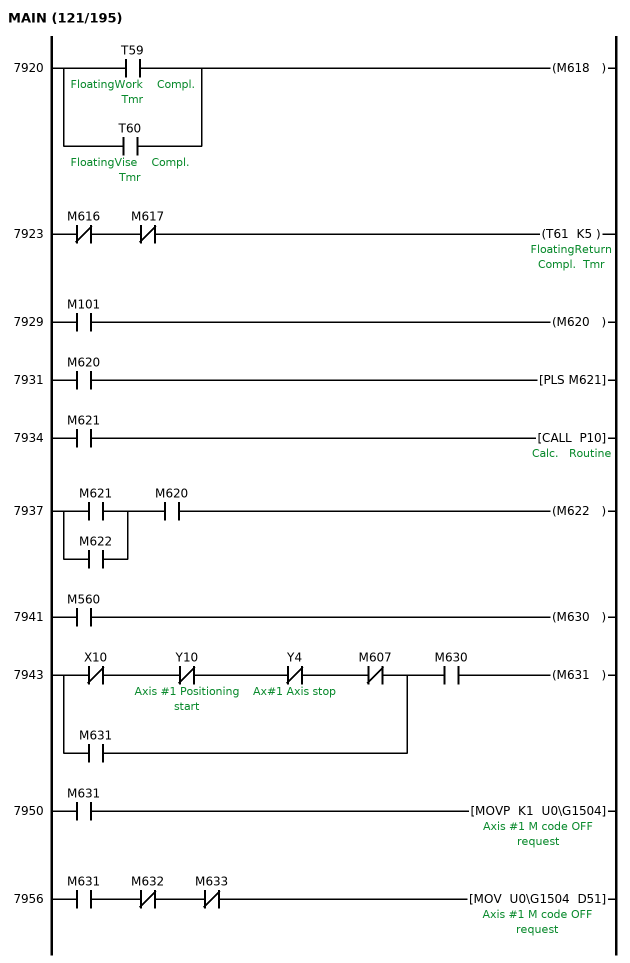
[picture p120: ladder of MAIN, rungs at steps 7920 to 7956]
7920  LD      T59  ; FloatingWork    Compl.  Tmr
      OR      T60  ; FloatingVise    Compl.  Tmr
      OUT     M618
7923  LDI     M616
      ANI     M617
      OUT     T61 K5  ; FloatingReturn  Compl.  Tmr
7929  LD      M101
      OUT     M620
7931  LD      M620
      PLS     M621
7934  LD      M621
      CALL    P10  ; Calc.   Routine
7937  LD      M621
      OR      M622
      AND     M620
      OUT     M622
7941  LD      M560
      OUT     M630
7943  LDI     X10
      ANI     Y10  ; Axis #1 Positioning start
      ANI     Y4  ; Ax#1 Axis stop
      ANI     M607
      OR      M631
      AND     M630
      OUT     M631
7950  LD      M631
      MOVP    K1 U0\G1504  ; Axis #1 M code OFF request
7956  LD      M631
      ANI     M632
      ANI     M633
      MOV     U0\G1504 D51
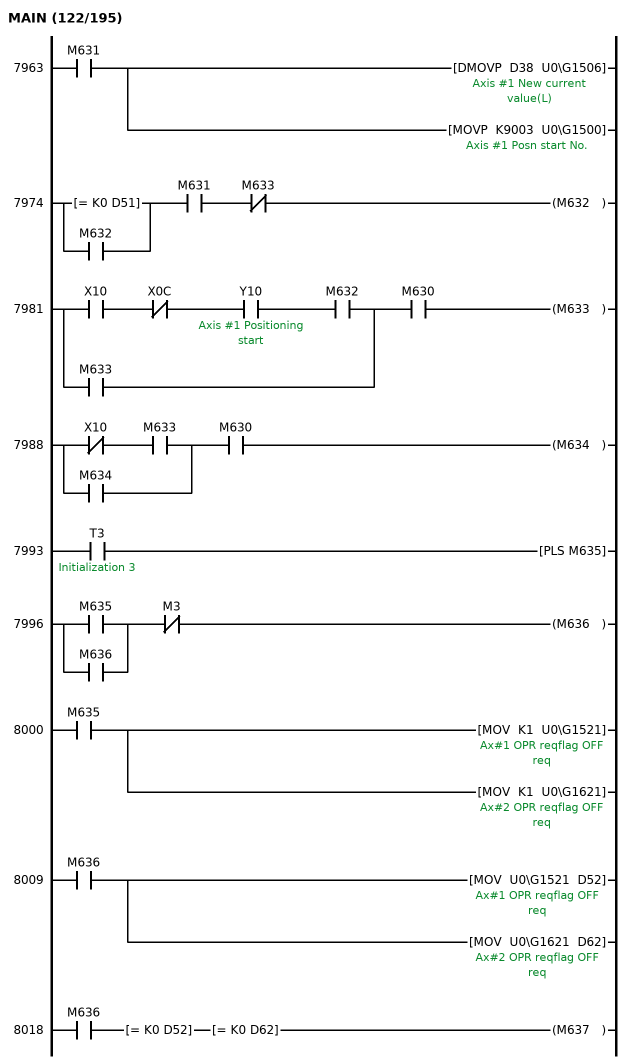
7963  LD      M631
      DMOVP   D38 U0\G1506  ; Axis #1 New current value(L)
      MOVP    K9003 U0\G1500
7974  LD=     K0 D51
      OR      M632
      AND     M631
      ANI     M633
      OUT     M632
7981  LD      X10
      ANI     X0C
      AND     Y10  ; Axis #1 Positioning start
      AND     M632
      OR      M633
      AND     M630
      OUT     M633
7988  LDI     X10
      AND     M633
      OR      M634
      AND     M630
      OUT     M634
7993  LD      T3  ; Initialization 3
      PLS     M635
7996  LD      M635
      OR      M636
      ANI     M3
      OUT     M636
8000  LD      M635
      MOV     K1 U0\G1521  ; Ax#1 OPR reqflag OFF req
      MOV     K1 U0\G1621  ; Ax#2 OPR reqflag OFF req
8009  LD      M636
      MOV     U0\G1521 D52
      MOV     U0\G1621 D62
8018  LD      M636
      AND=    K0 D52
      AND=    K0 D62
      OUT     M637
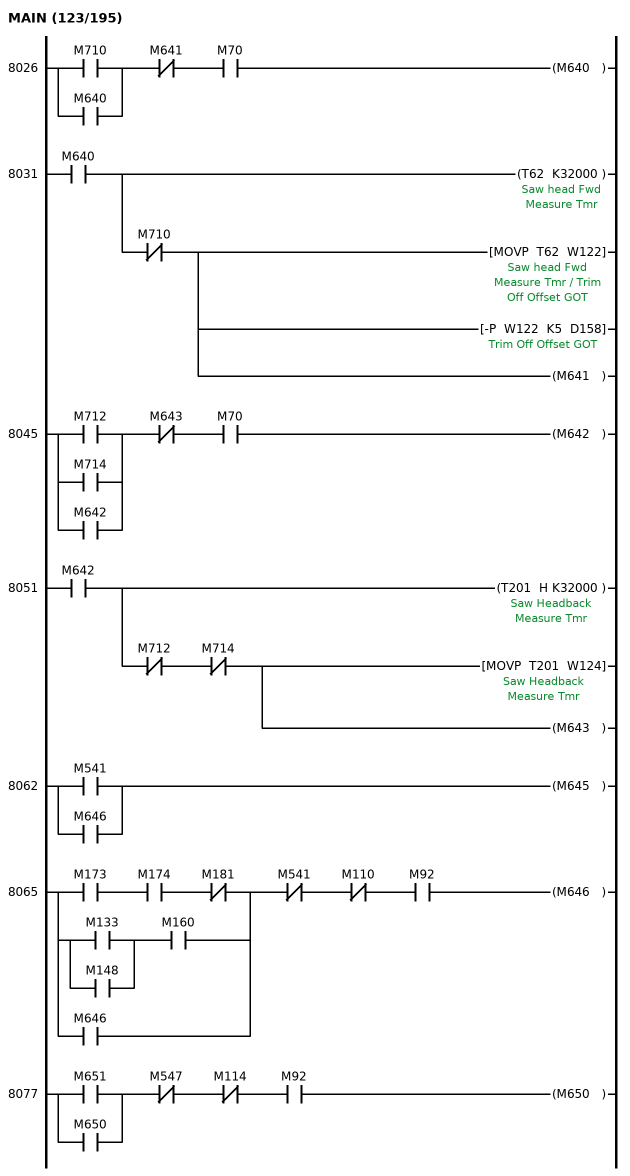
8026  LD      M710
      OR      M640
      ANI     M641
      AND     M70
      OUT     M640
8031  LD      M640
      OUT     T62 K32000  ; Saw head Fwd    Measure Tmr
      ANI     M710
      MOVP    T62 W122  ; Trim Off Offset GOT
      -P      W122 K5 D158
      OUT     M641
8045  LD      M712
      OR      M714
      OR      M642
      ANI     M643
      AND     M70
      OUT     M642
8051  LD      M642
      OUTH    T201 K32000  ; Saw Headback    Measure Tmr
      ANI     M712
      ANI     M714
      MOVP    T201 W124
      OUT     M643
8062  LD      M541
      OR      M646
      OUT     M645
8065  LD      M173
      AND     M174
      ANI     M181
      LD      M133
      OR      M148
      AND     M160
      ORB
      OR      M646
      ANI     M541
      ANI     M110
      AND     M92
      OUT     M646
8077  LD      M651
      OR      M650
      ANI     M547
      ANI     M114
      AND     M92
      OUT     M650
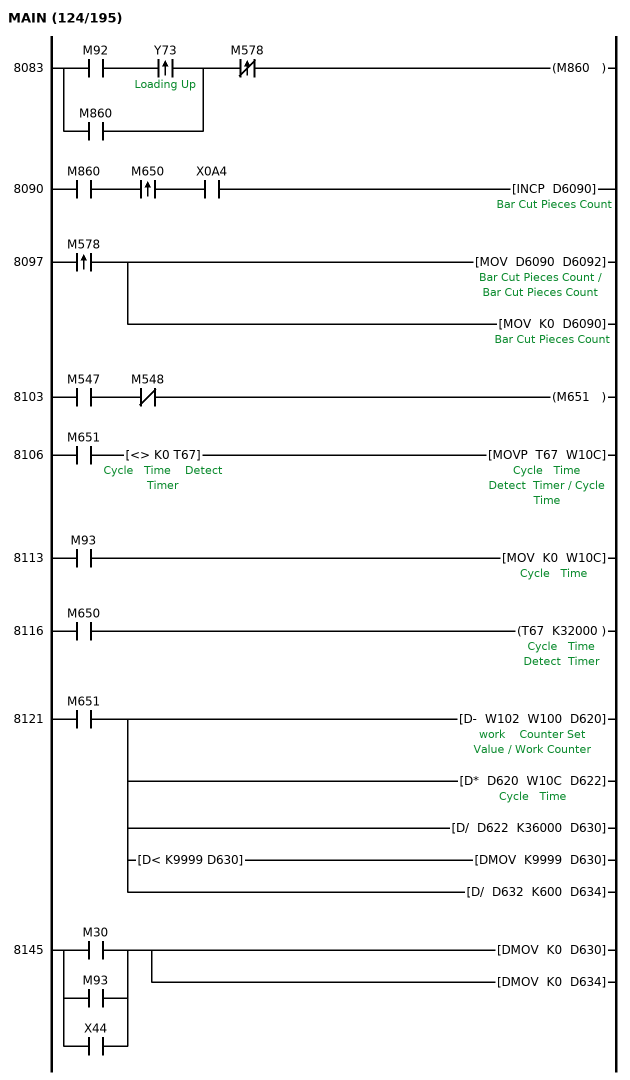
8083  LD      M92
      ANDP    Y73  ; Loading Up
      OR      M860
      ANDPI   M578
      OUT     M860
8090  LD      M860
      ANDP    M650
      AND     X0A4
      INCP    D6090  ; Bar Cut Pieces Count
8097  LDP     M578
      MOV     D6090 D6092  ; Bar Cut Pieces Count
      MOV     K0 D6090
8103  LD      M547
      ANI     M548
      OUT     M651
8106  LD      M651
      AND<>   K0 T67  ; Cycle   Time    Detect  Timer
      MOVP    T67 W10C  ; Cycle   Time
8113  LD      M93
      MOV     K0 W10C
8116  LD      M650
      OUT     T67 K32000  ; Cycle   Time    Detect  Timer
8121  LD      M651
      D-      W102 W100 D620
      D*      D620 W10C D622
      D/      D622 K36000 D630
      MPS
      ANDD<   K9999 D630
      DMOV    K9999 D630
      MPP
      D/      D632 K600 D634
8145  LD      M30
      OR      M93
      OR      X44
      DMOV    K0 D630
      DMOV    K0 D634
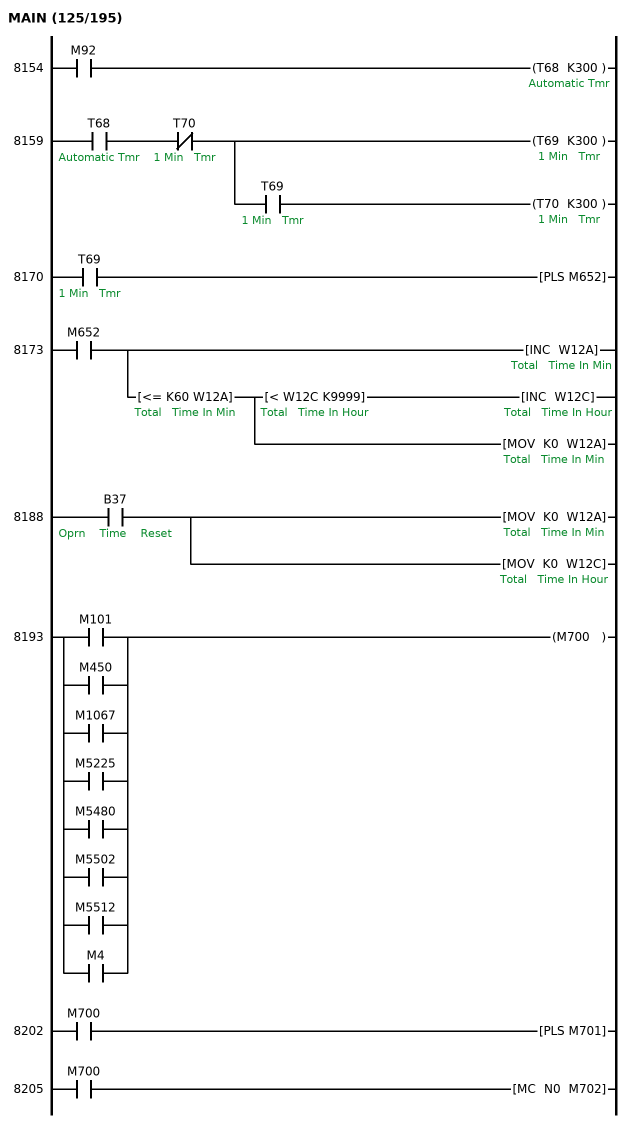
8154  LD      M92
      OUT     T68 K300  ; Automatic Tmr
8159  LD      T68  ; Automatic Tmr
      ANI     T70  ; 1 Min   Tmr
      OUT     T69 K300  ; 1 Min   Tmr
      AND     T69  ; 1 Min   Tmr
      OUT     T70 K300  ; 1 Min   Tmr
8170  LD      T69  ; 1 Min   Tmr
      PLS     M652
8173  LD      M652
      INC     W12A  ; Total   Time In Min
      AND<=   K60 W12A  ; Total   Time In Min
      MPS
      AND<    W12C K9999  ; Total   Time In Hour
      INC     W12C
      MPP
      MOV     K0 W12A
8188  LD      B37  ; Oprn    Time    Reset
      MOV     K0 W12A
      MOV     K0 W12C
8193  LD      M101
      OR      M450
      OR      M1067
      OR      M5225
      OR      M5480
      OR      M5502
      OR      M5512
      OR      M4
      OUT     M700
8202  LD      M700
      PLS     M701
8205  LD      M700
      MC      N0 M702
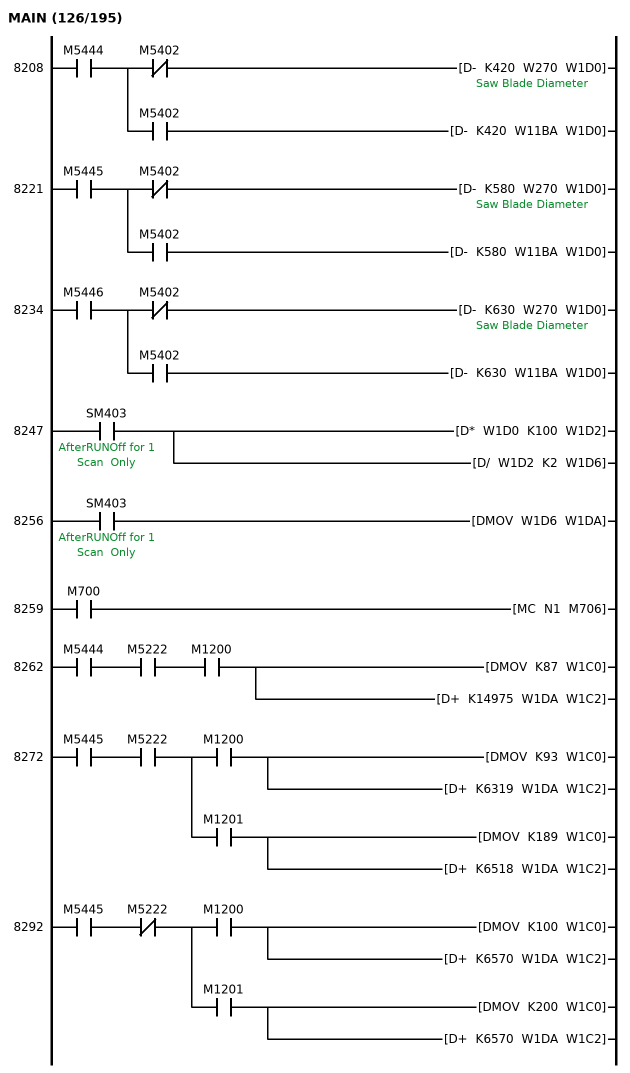
8208  LD      M5444
      MPS
      ANI     M5402
      D-      K420 W270 W1D0
      MPP
      AND     M5402
      D-      K420 W11BA W1D0
8221  LD      M5445
      MPS
      ANI     M5402
      D-      K580 W270 W1D0
      MPP
      AND     M5402
      D-      K580 W11BA W1D0
8234  LD      M5446
      MPS
      ANI     M5402
      D-      K630 W270 W1D0
      MPP
      AND     M5402
      D-      K630 W11BA W1D0
8247  LD      SM403  ; AfterRUNOff for 1 Scan  Only
      D*      W1D0 K100 W1D2
      D/      W1D2 K2 W1D6
8256  LD      SM403  ; AfterRUNOff for 1 Scan  Only
      DMOV    W1D6 W1DA
8259  LD      M700
      MC      N1 M706
8262  LD      M5444
      AND     M5222
      AND     M1200
      DMOV    K87 W1C0
      D+      K14975 W1DA W1C2
8272  LD      M5445
      AND     M5222
      MPS
      AND     M1200
      DMOV    K93 W1C0
      D+      K6319 W1DA W1C2
      MPP
      AND     M1201
      DMOV    K189 W1C0
      D+      K6518 W1DA W1C2
8292  LD      M5445
      ANI     M5222
      MPS
      AND     M1200
      DMOV    K100 W1C0
      D+      K6570 W1DA W1C2
      MPP
      AND     M1201
      DMOV    K200 W1C0
      D+      K6570 W1DA W1C2
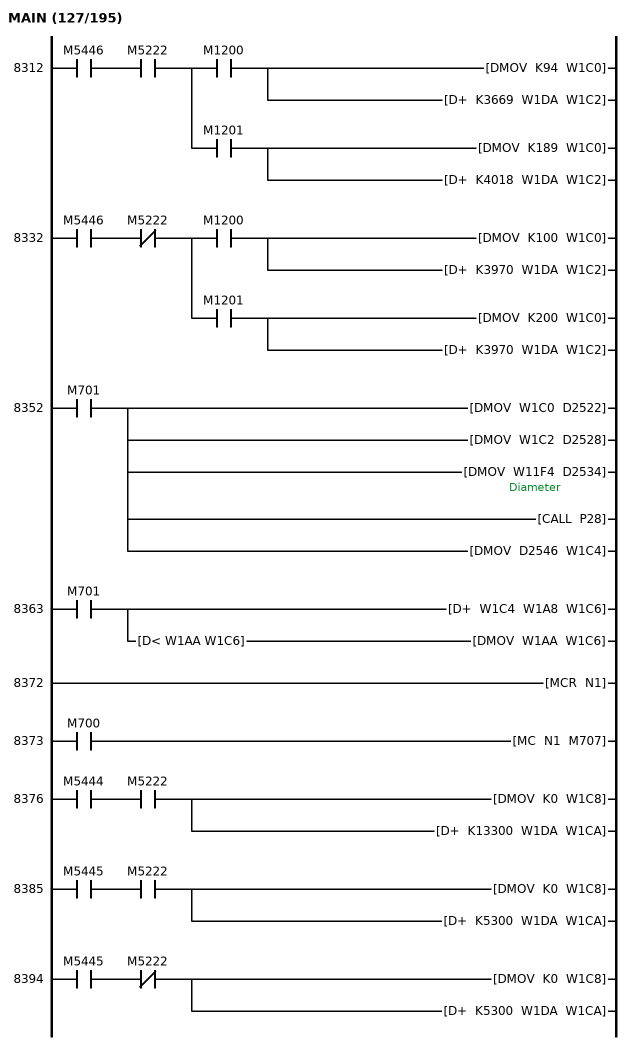
8312  LD      M5446
      AND     M5222
      MPS
      AND     M1200
      DMOV    K94 W1C0
      D+      K3669 W1DA W1C2
      MPP
      AND     M1201
      DMOV    K189 W1C0
      D+      K4018 W1DA W1C2
8332  LD      M5446
      ANI     M5222
      MPS
      AND     M1200
      DMOV    K100 W1C0
      D+      K3970 W1DA W1C2
      MPP
      AND     M1201
      DMOV    K200 W1C0
      D+      K3970 W1DA W1C2
8352  LD      M701
      DMOV    W1C0 D2522
      DMOV    W1C2 D2528
      DMOV    W11F4 D2534
      CALL    P28
      DMOV    D2546 W1C4
8363  LD      M701
      D+      W1C4 W1A8 W1C6
      ANDD<   W1AA W1C6
      DMOV    W1AA W1C6
8372  MCR     N1
8373  LD      M700
      MC      N1 M707
8376  LD      M5444
      AND     M5222
      DMOV    K0 W1C8
      D+      K13300 W1DA W1CA
8385  LD      M5445
      AND     M5222
      DMOV    K0 W1C8
      D+      K5300 W1DA W1CA
8394  LD      M5445
      ANI     M5222
      DMOV    K0 W1C8
      D+      K5300 W1DA W1CA
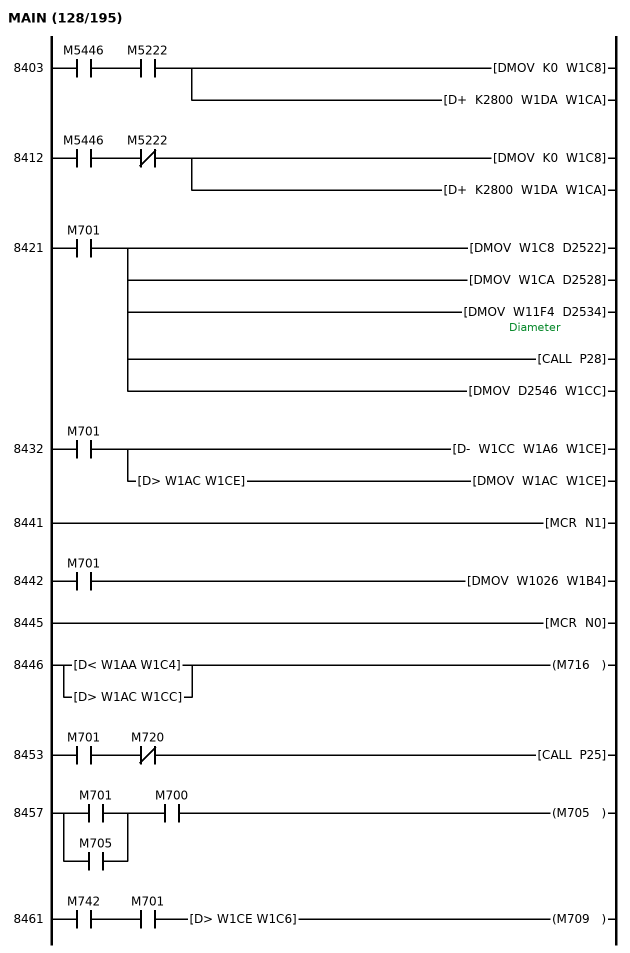
8403  LD      M5446
      AND     M5222
      DMOV    K0 W1C8
      D+      K2800 W1DA W1CA
8412  LD      M5446
      ANI     M5222
      DMOV    K0 W1C8
      D+      K2800 W1DA W1CA
8421  LD      M701
      DMOV    W1C8 D2522
      DMOV    W1CA D2528
      DMOV    W11F4 D2534
      CALL    P28
      DMOV    D2546 W1CC
8432  LD      M701
      D-      W1CC W1A6 W1CE
      ANDD>   W1AC W1CE
      DMOV    W1AC W1CE
8441  MCR     N1
8442  LD      M701
      DMOV    W1026 W1B4
8445  MCR     N0
8446  LDD<    W1AA W1C4
      ORD>    W1AC W1CC
      OUT     M716
8453  LD      M701
      ANI     M720
      CALL    P25
8457  LD      M701
      OR      M705
      AND     M700
      OUT     M705
8461  LD      M742
      AND     M701
      ANDD>   W1CE W1C6
      OUT     M709
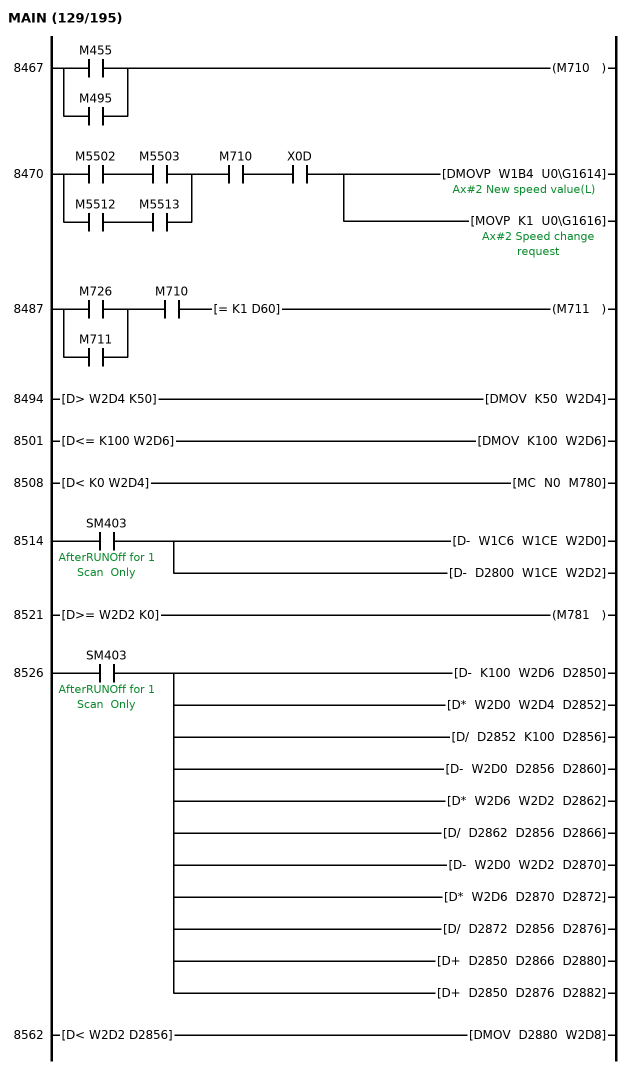
8467  LD      M455
      OR      M495
      OUT     M710
8470  LD      M5502
      AND     M5503
      LD      M5512
      AND     M5513
      ORB
      AND     M710
      AND     X0D
      DMOVP   W1B4 U0\G1614  ; Ax#2 New speed value(L)
      MOVP    K1 U0\G1616  ; Ax#2 Speed change request
8487  LD      M726
      OR      M711
      AND     M710
      AND=    K1 D60
      OUT     M711
8494  LDD>    W2D4 K50
      DMOV    K50 W2D4
8501  LDD<=   K100 W2D6
      DMOV    K100 W2D6
8508  LDD<    K0 W2D4
      MC      N0 M780
8514  LD      SM403  ; AfterRUNOff for 1 Scan  Only
      D-      W1C6 W1CE W2D0
      D-      D2800 W1CE W2D2
8521  LDD>=   W2D2 K0
      OUT     M781
8526  LD      SM403  ; AfterRUNOff for 1 Scan  Only
      D-      K100 W2D6 D2850
      D*      W2D0 W2D4 D2852
      D/      D2852 K100 D2856
      D-      W2D0 D2856 D2860
      D*      W2D6 W2D2 D2862
      D/      D2862 D2856 D2866
      D-      W2D0 W2D2 D2870
      D*      W2D6 D2870 D2872
      D/      D2872 D2856 D2876
      D+      D2850 D2866 D2880
      D+      D2850 D2876 D2882
8562  LDD<    W2D2 D2856
      DMOV    D2880 W2D8
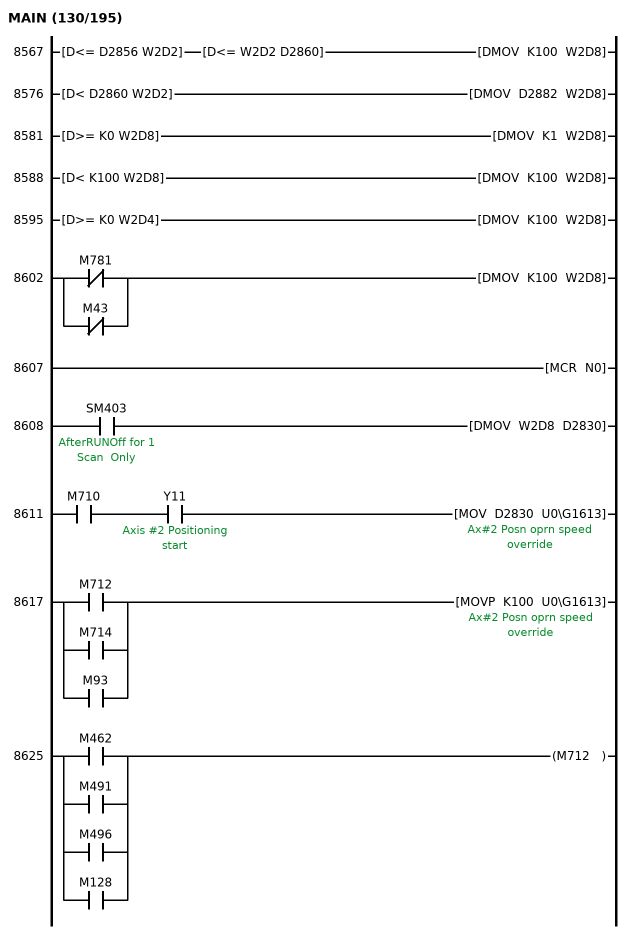
8567  LDD<=   D2856 W2D2
      ANDD<=  W2D2 D2860
      DMOV    K100 W2D8
8576  LDD<    D2860 W2D2
      DMOV    D2882 W2D8
8581  LDD>=   K0 W2D8
      DMOV    K1 W2D8
8588  LDD<    K100 W2D8
      DMOV    K100 W2D8
8595  LDD>=   K0 W2D4
      DMOV    K100 W2D8
8602  LDI     M781
      ORI     M43
      DMOV    K100 W2D8
8607  MCR     N0
8608  LD      SM403  ; AfterRUNOff for 1 Scan  Only
      DMOV    W2D8 D2830
8611  LD      M710
      AND     Y11  ; Axis #2 Positioning start
      MOV     D2830 U0\G1613  ; Ax#2 Posn oprn speed override
8617  LD      M712
      OR      M714
      OR      M93
      MOVP    K100 U0\G1613
8625  LD      M462
      OR      M491
      OR      M496
      OR      M128
      OUT     M712
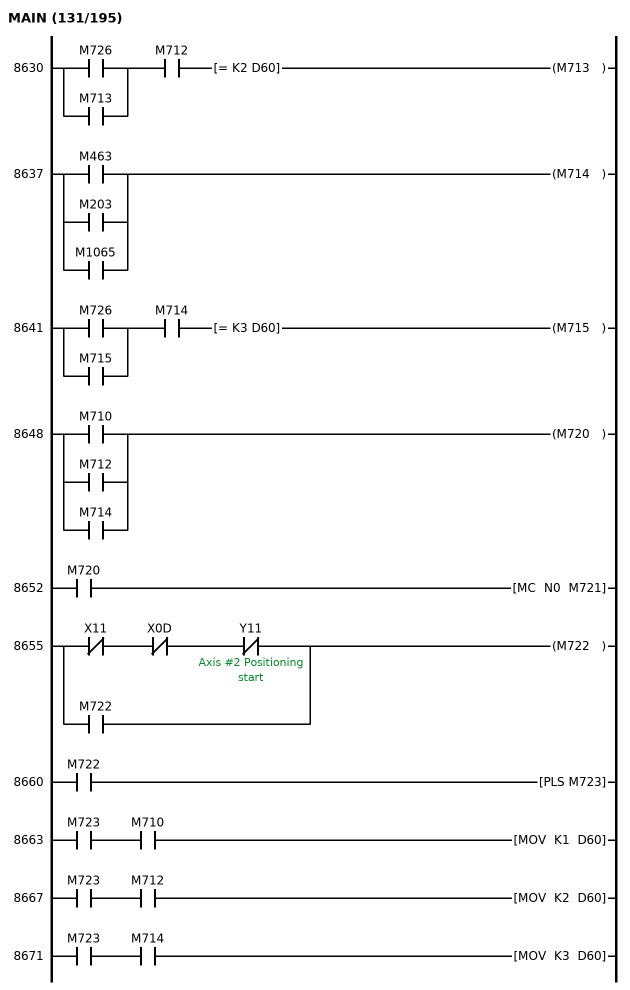
8630  LD      M726
      OR      M713
      AND     M712
      AND=    K2 D60
      OUT     M713
8637  LD      M463
      OR      M203
      OR      M1065
      OUT     M714
8641  LD      M726
      OR      M715
      AND     M714
      AND=    K3 D60
      OUT     M715
8648  LD      M710
      OR      M712
      OR      M714
      OUT     M720
8652  LD      M720
      MC      N0 M721
8655  LDI     X11
      ANI     X0D
      ANI     Y11  ; Axis #2 Positioning start
      OR      M722
      OUT     M722
8660  LD      M722
      PLS     M723
8663  LD      M723
      AND     M710
      MOV     K1 D60
8667  LD      M723
      AND     M712
      MOV     K2 D60
8671  LD      M723
      AND     M714
      MOV     K3 D60
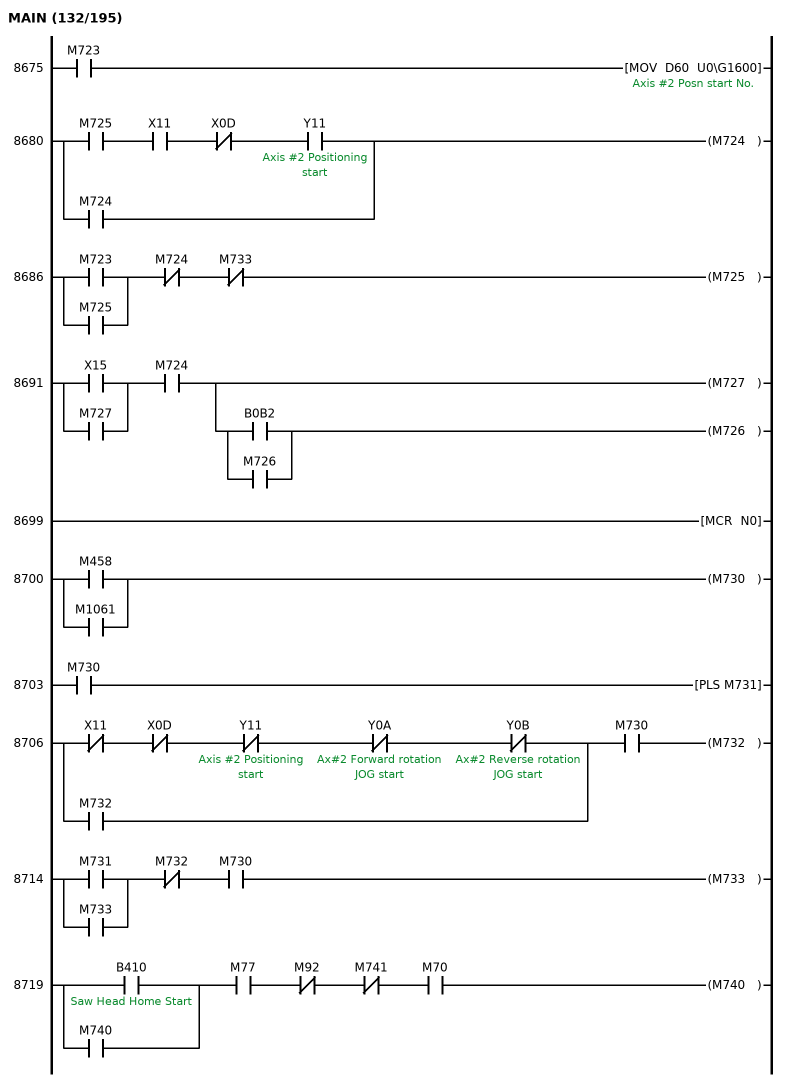
8675  LD      M723
      MOV     D60 U0\G1600  ; Axis #2 Posn start No.
8680  LD      M725
      AND     X11
      ANI     X0D
      AND     Y11  ; Axis #2 Positioning start
      OR      M724
      OUT     M724
8686  LD      M723
      OR      M725
      ANI     M724
      ANI     M733
      OUT     M725
8691  LD      X15
      OR      M727
      AND     M724
      OUT     M727
      LD      B0B2
      OR      M726
      ANB
      OUT     M726
8699  MCR     N0
8700  LD      M458
      OR      M1061
      OUT     M730
8703  LD      M730
      PLS     M731
8706  LDI     X11
      ANI     X0D
      ANI     Y11  ; Axis #2 Positioning start
      ANI     Y0A  ; Ax#2 Forward rotation JOG start
      ANI     Y0B  ; Ax#2 Reverse rotation JOG start
      OR      M732
      AND     M730
      OUT     M732
8714  LD      M731
      OR      M733
      ANI     M732
      AND     M730
      OUT     M733
8719  LD      B410  ; Saw Head Home Start
      OR      M740
      AND     M77
      ANI     M92
      ANI     M741
      AND     M70
      OUT     M740
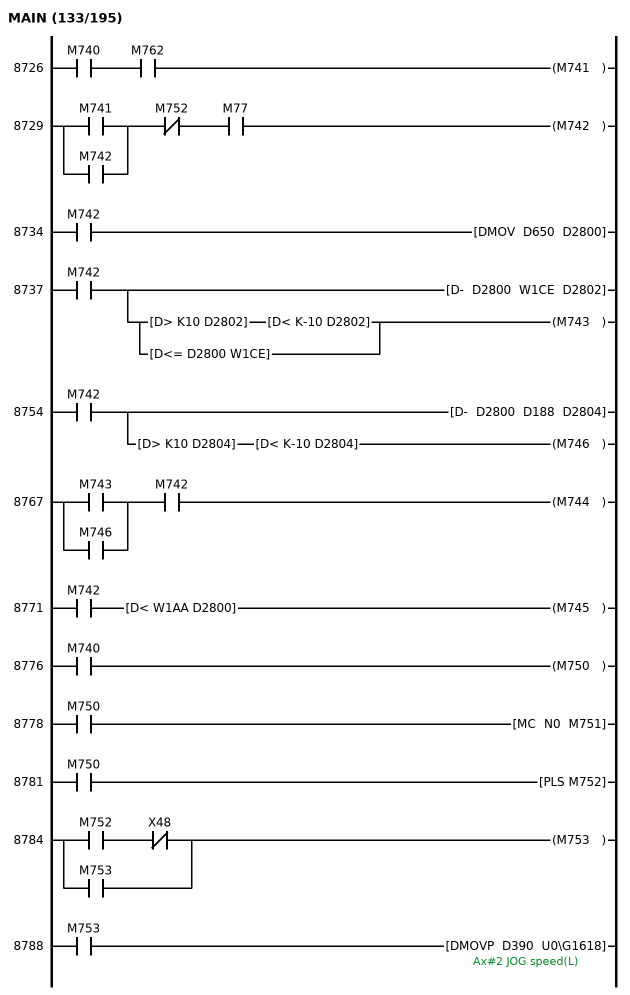
8726  LD      M740
      AND     M762
      OUT     M741
8729  LD      M741
      OR      M742
      ANI     M752
      AND     M77
      OUT     M742
8734  LD      M742
      DMOV    D650 D2800
8737  LD      M742
      D-      D2800 W1CE D2802
      LDD>    K10 D2802
      ANDD<   K-10 D2802
      ORD<=   D2800 W1CE
      ANB
      OUT     M743
8754  LD      M742
      D-      D2800 D188 D2804
      ANDD>   K10 D2804
      ANDD<   K-10 D2804
      OUT     M746
8767  LD      M743
      OR      M746
      AND     M742
      OUT     M744
8771  LD      M742
      ANDD<   W1AA D2800
      OUT     M745
8776  LD      M740
      OUT     M750
8778  LD      M750
      MC      N0 M751
8781  LD      M750
      PLS     M752
8784  LD      M752
      ANI     X48
      OR      M753
      OUT     M753
8788  LD      M753
      DMOVP   D390 U0\G1618
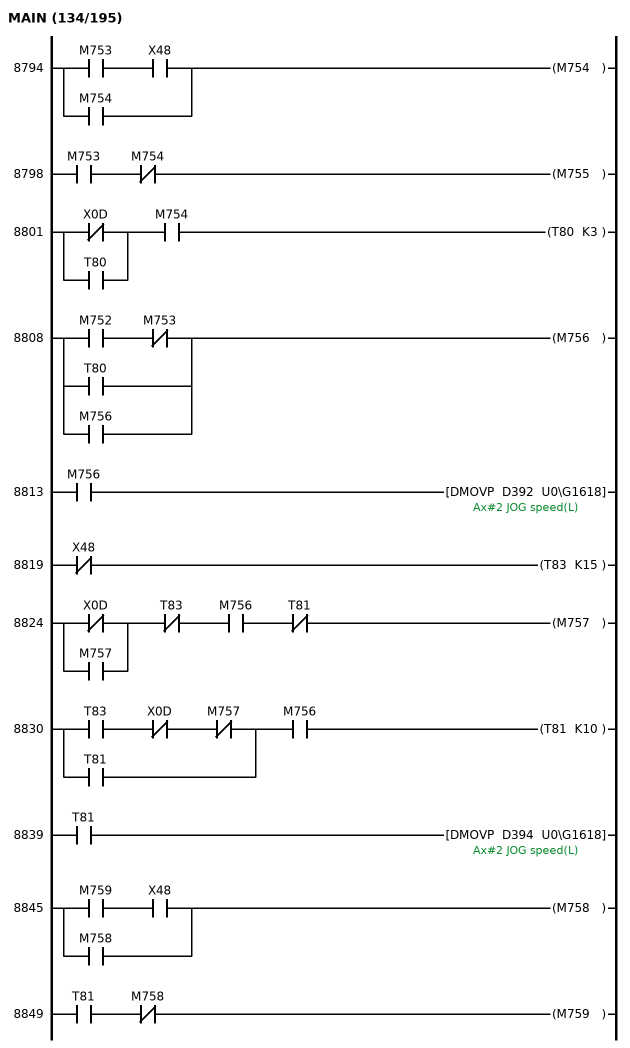
8794  LD      M753
      AND     X48
      OR      M754
      OUT     M754
8798  LD      M753
      ANI     M754
      OUT     M755
8801  LDI     X0D
      OR      T80
      AND     M754
      OUT     T80 K3
8808  LD      M752
      ANI     M753
      OR      T80
      OR      M756
      OUT     M756
8813  LD      M756
      DMOVP   D392 U0\G1618
8819  LDI     X48
      OUT     T83 K15
8824  LDI     X0D
      OR      M757
      ANI     T83
      AND     M756
      ANI     T81
      OUT     M757
8830  LD      T83
      ANI     X0D
      ANI     M757
      OR      T81
      AND     M756
      OUT     T81 K10
8839  LD      T81
      DMOVP   D394 U0\G1618
8845  LD      M759
      AND     X48
      OR      M758
      OUT     M758
8849  LD      T81
      ANI     M758
      OUT     M759
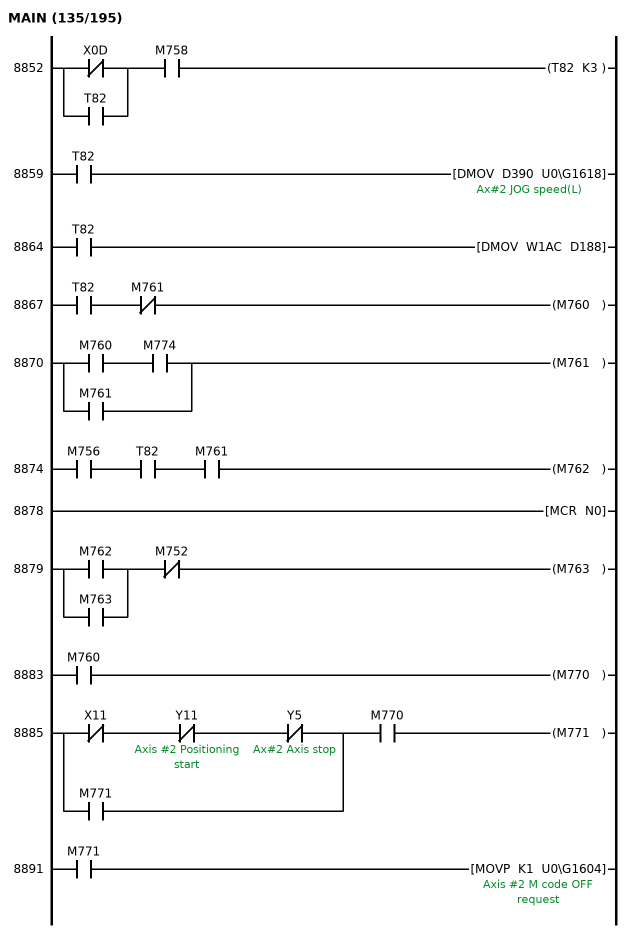
8852  LDI     X0D
      OR      T82
      AND     M758
      OUT     T82 K3
8859  LD      T82
      DMOV    D390 U0\G1618
8864  LD      T82
      DMOV    W1AC D188
8867  LD      T82
      ANI     M761
      OUT     M760
8870  LD      M760
      AND     M774
      OR      M761
      OUT     M761
8874  LD      M756
      AND     T82
      AND     M761
      OUT     M762
8878  MCR     N0
8879  LD      M762
      OR      M763
      ANI     M752
      OUT     M763
8883  LD      M760
      OUT     M770
8885  LDI     X11
      ANI     Y11  ; Axis #2 Positioning start
      ANI     Y5  ; Ax#2 Axis stop
      OR      M771
      AND     M770
      OUT     M771
8891  LD      M771
      MOVP    K1 U0\G1604  ; Axis #2 M code OFF request
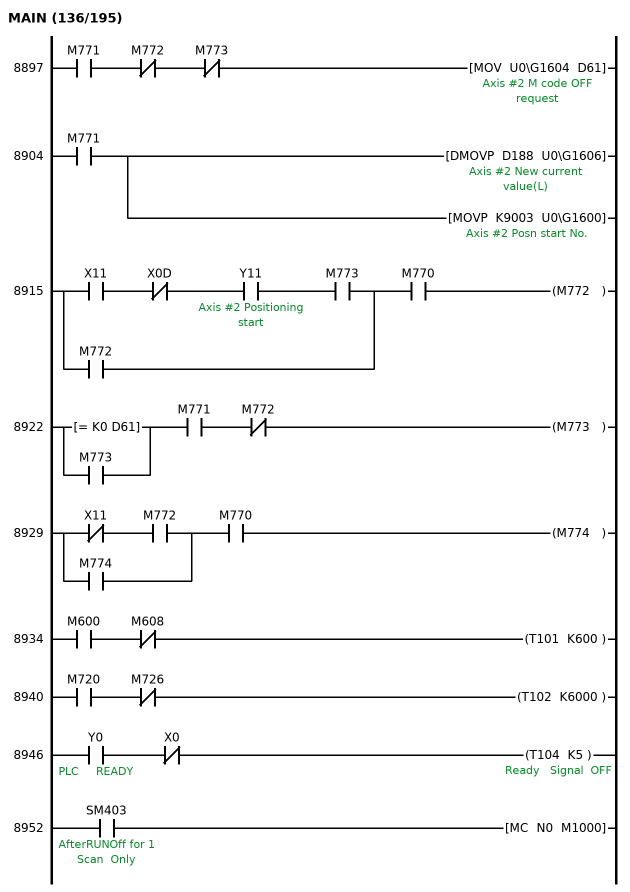
8897  LD      M771
      ANI     M772
      ANI     M773
      MOV     U0\G1604 D61
8904  LD      M771
      DMOVP   D188 U0\G1606  ; Axis #2 New current value(L)
      MOVP    K9003 U0\G1600
8915  LD      X11
      ANI     X0D
      AND     Y11  ; Axis #2 Positioning start
      AND     M773
      OR      M772
      AND     M770
      OUT     M772
8922  LD=     K0 D61
      OR      M773
      AND     M771
      ANI     M772
      OUT     M773
8929  LDI     X11
      AND     M772
      OR      M774
      AND     M770
      OUT     M774
8934  LD      M600
      ANI     M608
      OUT     T101 K600
8940  LD      M720
      ANI     M726
      OUT     T102 K6000
8946  LD      Y0  ; PLC     READY
      ANI     X0
      OUT     T104 K5  ; Ready   Signal  OFF
8952  LD      SM403  ; AfterRUNOff for 1 Scan  Only
      MC      N0 M1000
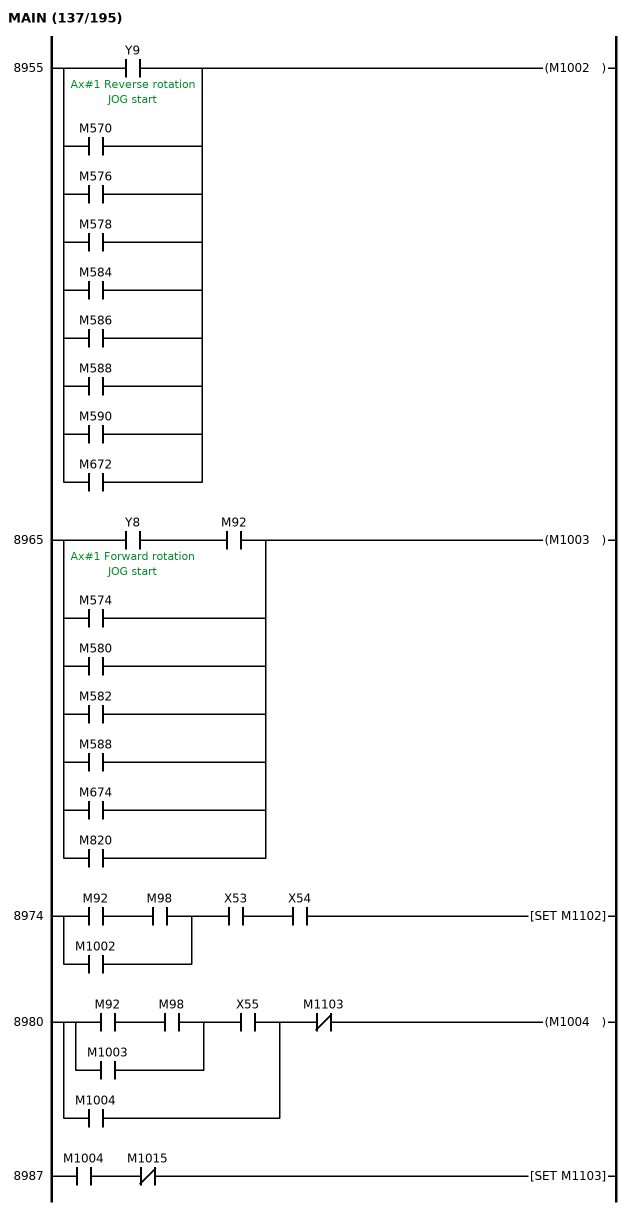
8955  LD      Y9  ; Ax#1 Reverse rotation JOG start
      OR      M570
      OR      M576
      OR      M578
      OR      M584
      OR      M586
      OR      M588
      OR      M590
      OR      M672
      OUT     M1002
8965  LD      Y8  ; Ax#1 Forward rotation JOG start
      AND     M92
      OR      M574
      OR      M580
      OR      M582
      OR      M588
      OR      M674
      OR      M820
      OUT     M1003
8974  LD      M92
      AND     M98
      OR      M1002
      AND     X53
      AND     X54
      SET     M1102
8980  LD      M92
      AND     M98
      OR      M1003
      AND     X55
      OR      M1004
      ANI     M1103
      OUT     M1004
8987  LD      M1004
      ANI     M1015
      SET     M1103
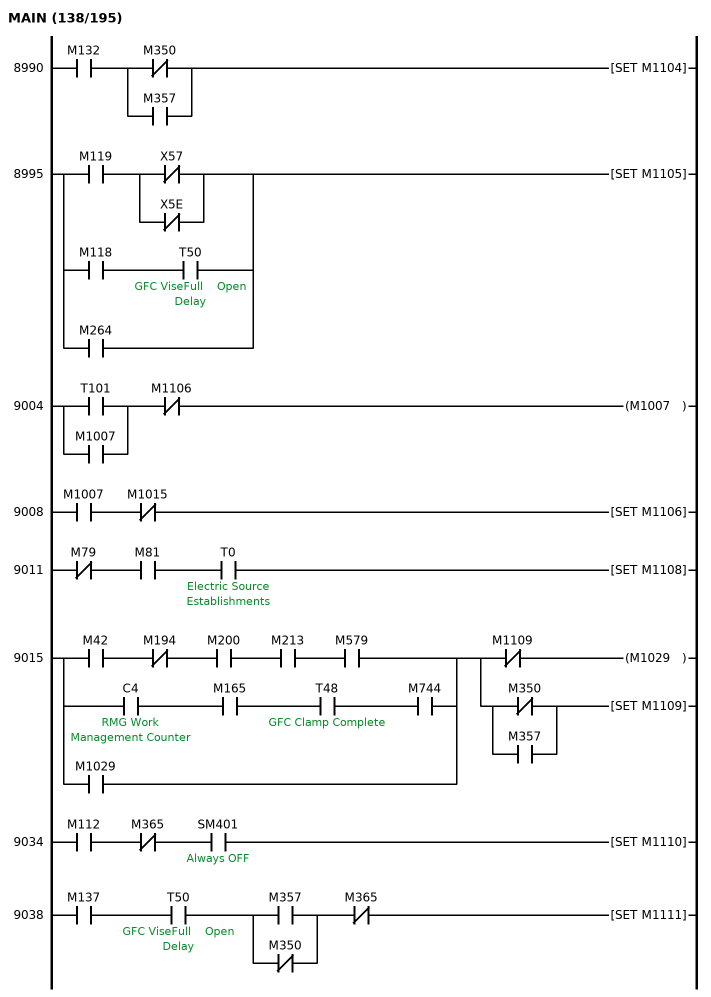
8990  LD      M132
      LDI     M350
      OR      M357
      ANB
      SET     M1104
8995  LD      M119
      LDI     X57
      ORI     X5E
      ANB
      LD      M118
      AND     T50  ; GFC ViseFull    Open    Delay
      ORB
      OR      M264
      SET     M1105
9004  LD      T101
      OR      M1007
      ANI     M1106
      OUT     M1007
9008  LD      M1007
      ANI     M1015
      SET     M1106
9011  LDI     M79
      AND     M81
      AND     T0  ; Electric Source Establishments
      SET     M1108
9015  LD      M42
      ANI     M194
      AND     M200
      AND     M213
      AND     M579
      LD      C4  ; RMG WorkManagement Counter
      AND     M165
      AND     T48  ; GFC Clamp Complete
      AND     M744
      ORB
      OR      M1029
      MPS
      ANI     M1109
      OUT     M1029
      MPP
      LDI     M350
      OR      M357
      ANB
      SET     M1109
9034  LD      M112
      ANI     M365
      AND     SM401  ; Always OFF
      SET     M1110
9038  LD      M137
      AND     T50  ; GFC ViseFull    Open    Delay
      LD      M357
      ORI     M350
      ANB
      ANI     M365
      SET     M1111
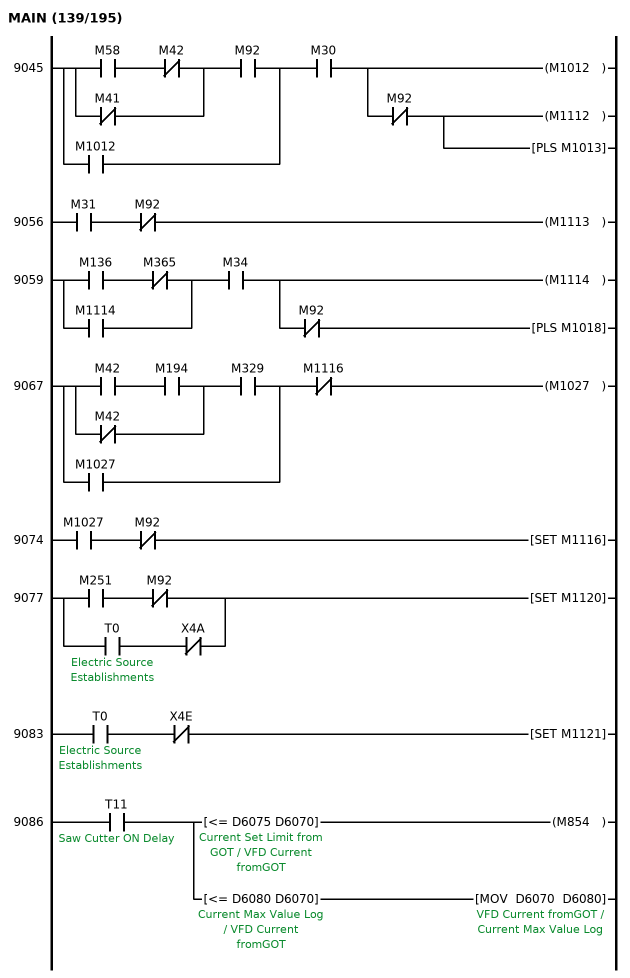
9045  LD      M58
      ANI     M42
      ORI     M41
      AND     M92
      OR      M1012
      AND     M30
      OUT     M1012
      ANI     M92
      OUT     M1112
      PLS     M1013
9056  LD      M31
      ANI     M92
      OUT     M1113
9059  LD      M136
      ANI     M365
      OR      M1114
      AND     M34
      OUT     M1114
      ANI     M92
      PLS     M1018
9067  LD      M42
      AND     M194
      ORI     M42
      AND     M329
      OR      M1027
      ANI     M1116
      OUT     M1027
9074  LD      M1027
      ANI     M92
      SET     M1116
9077  LD      M251
      ANI     M92
      LD      T0  ; Electric Source Establishments
      ANI     X4A
      ORB
      SET     M1120
9083  LD      T0  ; Electric Source Establishments
      ANI     X4E
      SET     M1121
9086  LD      T11  ; Saw Cutter ON Delay
      MPS
      AND<=   D6075 D6070  ; Current Set Limit from GOT / VFD Current fromGOT
      OUT     M854
      MPP
      AND<=   D6080 D6070  ; Current Max Value Log / VFD Current fromGOT
      MOV     D6070 D6080
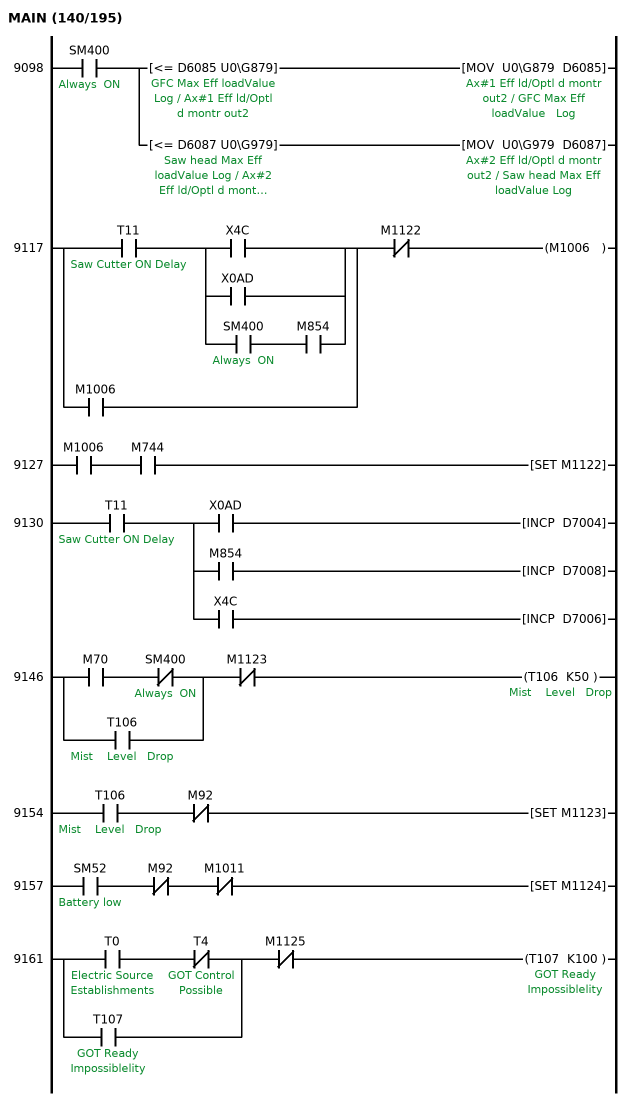
9098  LD      SM400  ; Always  ON
      MPS
      AND<=   D6085 U0\G879  ; GFC Max Eff loadValue   Log / Ax#1 Eff ld/Optl d montr out2
      MOV     U0\G879 D6085
      MPP
      AND<=   D6087 U0\G979  ; Saw head Max Eff loadValue Log / Ax#2 Eff ld/Optl d montr out2
      MOV     U0\G979 D6087
9117  LD      T11  ; Saw Cutter ON Delay
      LD      X4C
      OR      X0AD
      LD      SM400  ; Always  ON
      AND     M854
      ORB
      ANB
      OR      M1006
      ANI     M1122
      OUT     M1006
9127  LD      M1006
      AND     M744
      SET     M1122
9130  LD      T11  ; Saw Cutter ON Delay
      MPS
      AND     X0AD
      INCP    D7004
      MRD
      AND     M854
      INCP    D7008
      MPP
      AND     X4C
      INCP    D7006
9146  LD      M70
      ANI     SM400  ; Always  ON
      OR      T106  ; Mist    Level   Drop
      ANI     M1123
      OUT     T106 K50  ; Mist    Level   Drop
9154  LD      T106  ; Mist    Level   Drop
      ANI     M92
      SET     M1123
9157  LD      SM52  ; Battery low
      ANI     M92
      ANI     M1011
      SET     M1124
9161  LD      T0  ; Electric Source Establishments
      ANI     T4  ; GOT Control     Possible
      OR      T107  ; GOT Ready Impossiblelity
      ANI     M1125
      OUT     T107 K100  ; GOT Ready Impossiblelity
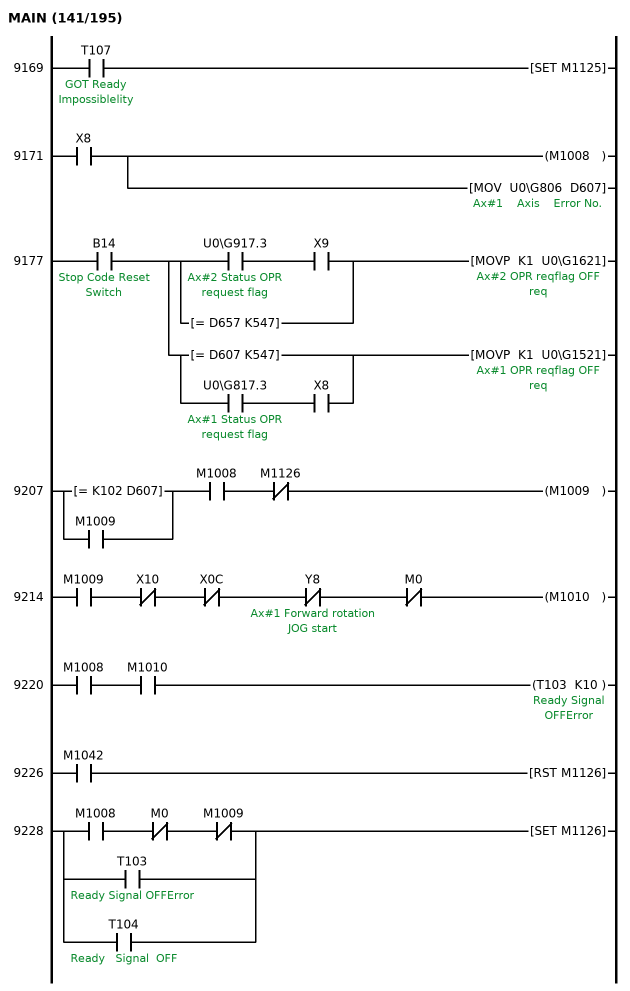
9169  LD      T107  ; GOT Ready Impossiblelity
      SET     M1125
9171  LD      X8
      OUT     M1008
      MOV     U0\G806 D607
9177  LD      B14  ; Stop Code Reset Switch
      MPS
      LD      U0\G917.3  ; Ax#2 Status OPR request flag
      AND     X9
      OR=     D657 K547
      ANB
      MOVP    K1 U0\G1621
      MPP
      LD=     D607 K547
      LD      U0\G817.3  ; Ax#1 Status OPR request flag
      AND     X8
      ORB
      ANB
      MOVP    K1 U0\G1521
9207  LD=     K102 D607
      OR      M1009
      AND     M1008
      ANI     M1126
      OUT     M1009
9214  LD      M1009
      ANI     X10
      ANI     X0C
      ANI     Y8  ; Ax#1 Forward rotation JOG start
      ANI     M0
      OUT     M1010
9220  LD      M1008
      AND     M1010
      OUT     T103 K10  ; Ready Signal OFFError
9226  LD      M1042
      RST     M1126
9228  LD      M1008
      ANI     M0
      ANI     M1009
      OR      T103  ; Ready Signal OFFError
      OR      T104  ; Ready   Signal  OFF
      SET     M1126
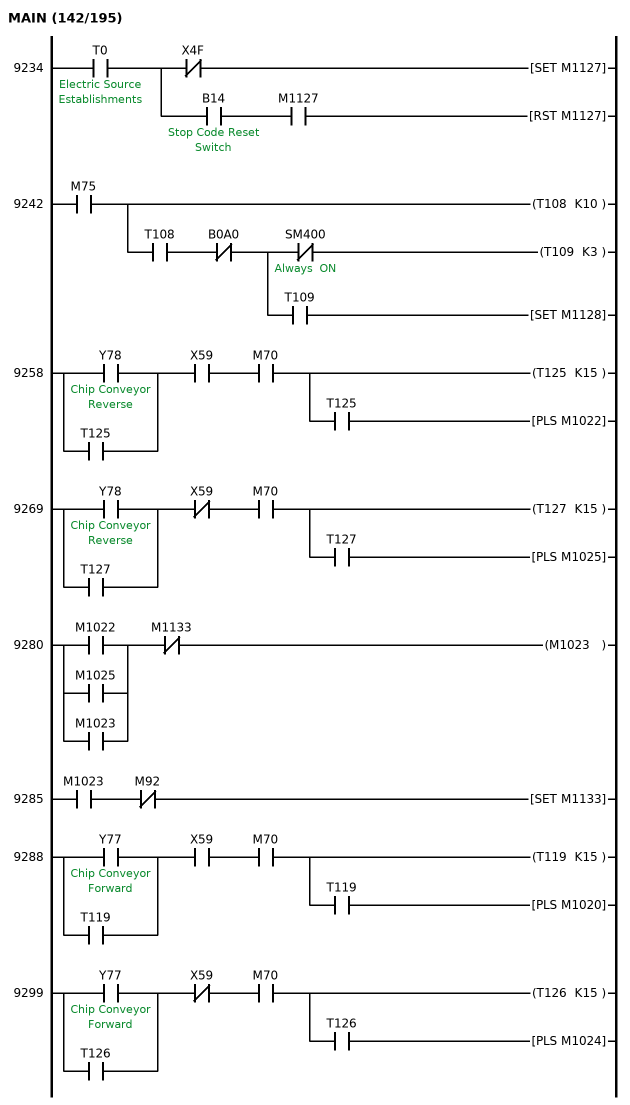
9234  LD      T0  ; Electric Source Establishments
      MPS
      ANI     X4F
      SET     M1127
      MPP
      AND     B14  ; Stop Code Reset Switch
      AND     M1127
      RST     M1127
9242  LD      M75
      OUT     T108 K10
      AND     T108
      ANI     B0A0
      MPS
      ANI     SM400  ; Always  ON
      OUT     T109 K3
      MPP
      AND     T109
      SET     M1128
9258  LD      Y78  ; Chip Conveyor Reverse
      OR      T125
      AND     X59
      AND     M70
      OUT     T125 K15
      AND     T125
      PLS     M1022
9269  LD      Y78  ; Chip Conveyor Reverse
      OR      T127
      ANI     X59
      AND     M70
      OUT     T127 K15
      AND     T127
      PLS     M1025
9280  LD      M1022
      OR      M1025
      OR      M1023
      ANI     M1133
      OUT     M1023
9285  LD      M1023
      ANI     M92
      SET     M1133
9288  LD      Y77  ; Chip Conveyor Forward
      OR      T119
      AND     X59
      AND     M70
      OUT     T119 K15
      AND     T119
      PLS     M1020
9299  LD      Y77  ; Chip Conveyor Forward
      OR      T126
      ANI     X59
      AND     M70
      OUT     T126 K15
      AND     T126
      PLS     M1024
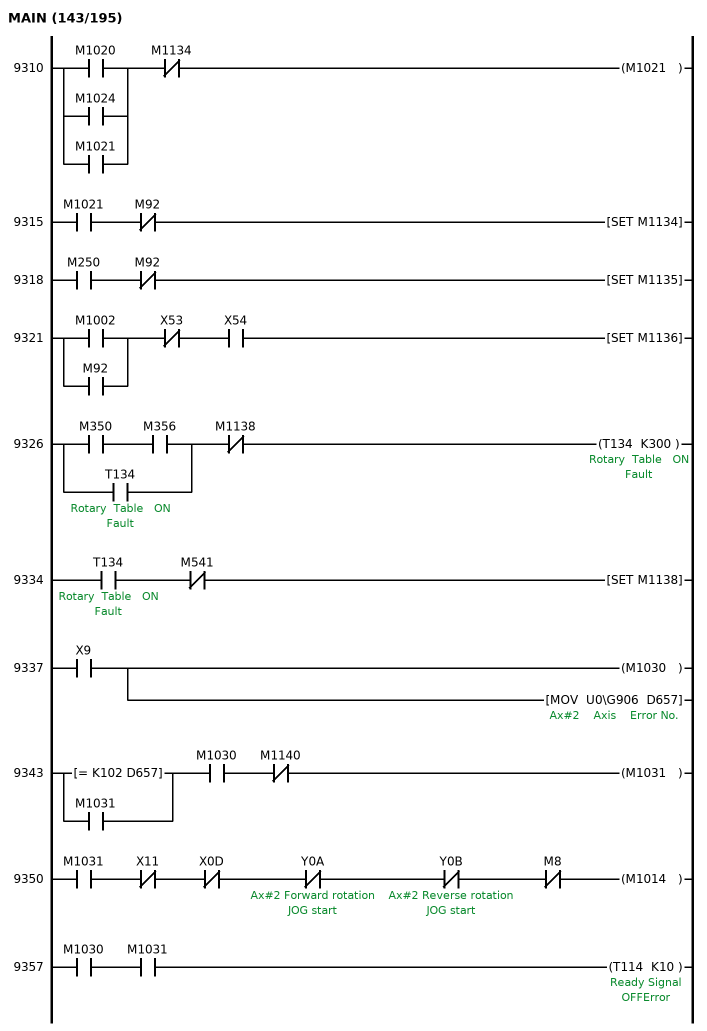
9310  LD      M1020
      OR      M1024
      OR      M1021
      ANI     M1134
      OUT     M1021
9315  LD      M1021
      ANI     M92
      SET     M1134
9318  LD      M250
      ANI     M92
      SET     M1135
9321  LD      M1002
      OR      M92
      ANI     X53
      AND     X54
      SET     M1136
9326  LD      M350
      AND     M356
      OR      T134  ; Rotary  Table   ON Fault
      ANI     M1138
      OUT     T134 K300  ; Rotary  Table   ON Fault
9334  LD      T134  ; Rotary  Table   ON Fault
      ANI     M541
      SET     M1138
9337  LD      X9
      OUT     M1030
      MOV     U0\G906 D657
9343  LD=     K102 D657
      OR      M1031
      AND     M1030
      ANI     M1140
      OUT     M1031
9350  LD      M1031
      ANI     X11
      ANI     X0D
      ANI     Y0A  ; Ax#2 Forward rotation JOG start
      ANI     Y0B  ; Ax#2 Reverse rotation JOG start
      ANI     M8
      OUT     M1014
9357  LD      M1030
      AND     M1031
      OUT     T114 K10  ; Ready Signal OFFError
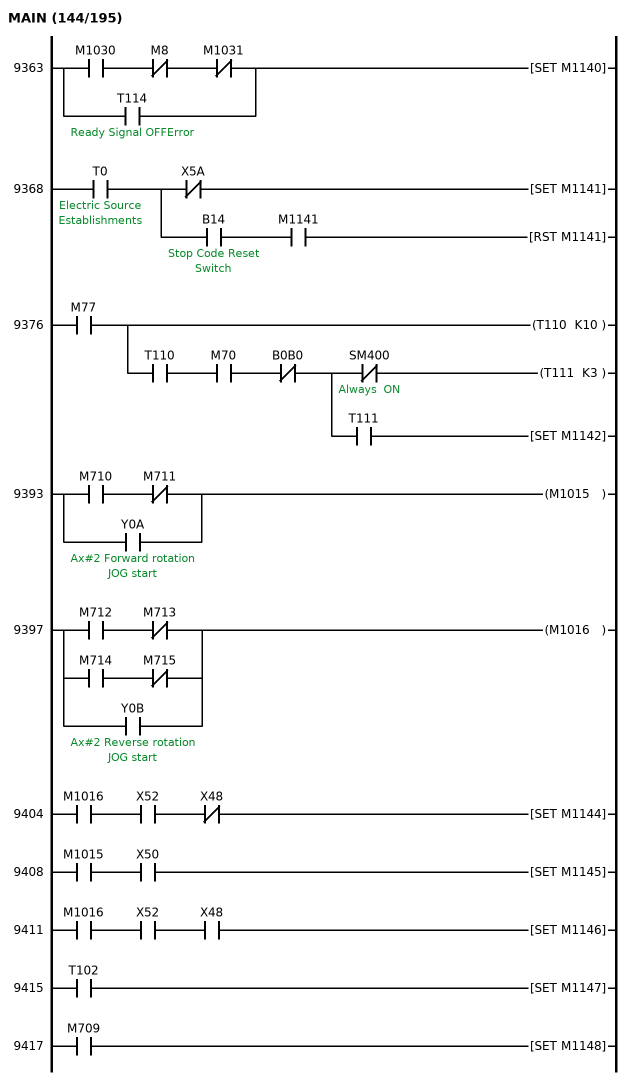
9363  LD      M1030
      ANI     M8
      ANI     M1031
      OR      T114  ; Ready Signal OFFError
      SET     M1140
9368  LD      T0  ; Electric Source Establishments
      MPS
      ANI     X5A
      SET     M1141
      MPP
      AND     B14  ; Stop Code Reset Switch
      AND     M1141
      RST     M1141
9376  LD      M77
      OUT     T110 K10
      AND     T110
      AND     M70
      ANI     B0B0
      MPS
      ANI     SM400  ; Always  ON
      OUT     T111 K3
      MPP
      AND     T111
      SET     M1142
9393  LD      M710
      ANI     M711
      OR      Y0A  ; Ax#2 Forward rotation JOG start
      OUT     M1015
9397  LD      M712
      ANI     M713
      LD      M714
      ANI     M715
      ORB
      OR      Y0B  ; Ax#2 Reverse rotation JOG start
      OUT     M1016
9404  LD      M1016
      AND     X52
      ANI     X48
      SET     M1144
9408  LD      M1015
      AND     X50
      SET     M1145
9411  LD      M1016
      AND     X52
      AND     X48
      SET     M1146
9415  LD      T102
      SET     M1147
9417  LD      M709
      SET     M1148
